FUNCTION_BLOCK FB_Calculator
VAR
END_VAR

METHOD Addition : LREAL;
VAR_INPUT
	a : LREAL;
	b : LREAL;
END_VAR
Addition := a + b;
END_METHOD

METHOD Substraction : LREAL
VAR_INPUT
	a : LREAL;
	b : LREAL;
END_VAR
Substraction := a - b;
END_METHOD

END_FUNCTION_BLOCK

(* stored: Version 1.1.0.1, ProductVersion 3.1.4024.14
   POU FB_Calculator: Id {d3162d3c-96b3-44be-be7e-6b3cbeb3741f}, SpecialFunc None
   Method Addition: Id {86bd279a-79ba-43c2-8260-1a47e17f6b05}
   Method Substraction: Id {38af8a8f-366e-41e9-842d-b208d9a90196} *)
